% RSLogix 500 project LEGACY PROGRAM NO LABELS ORIGINAL_BAK006.RSS, saved by version 11.00.00.00 %
PROJECT "ML1200"    % processor: MicroLogix 1200; MAIN_PROG %

PROGRAM FILES
  LAD 2 "MAIN_PROG"  15 rungs
  LAD 3   18 rungs
  LAD 4   33 rungs
  LAD 5   12 rungs
  LAD 6   14 rungs
  LAD 7   2 rungs
  LAD 8   47 rungs
  LAD 9   2 rungs
  LAD 10   5 rungs
  LAD 11   14 rungs

DATA FILES
  O0 OUTPUT  8 elements
  I1 INPUT  19 elements
  S2 STATUS  66 elements
  B3 BINARY  20 elements
  T4 TIMER  13 elements
  C5 COUNTER  1 elements
  R6 CONTROL  1 elements
  N7 INTEGER  77 elements
  F8 FLOAT  1 elements
  PD9   3 elements

LADDER 2 "MAIN_PROG"
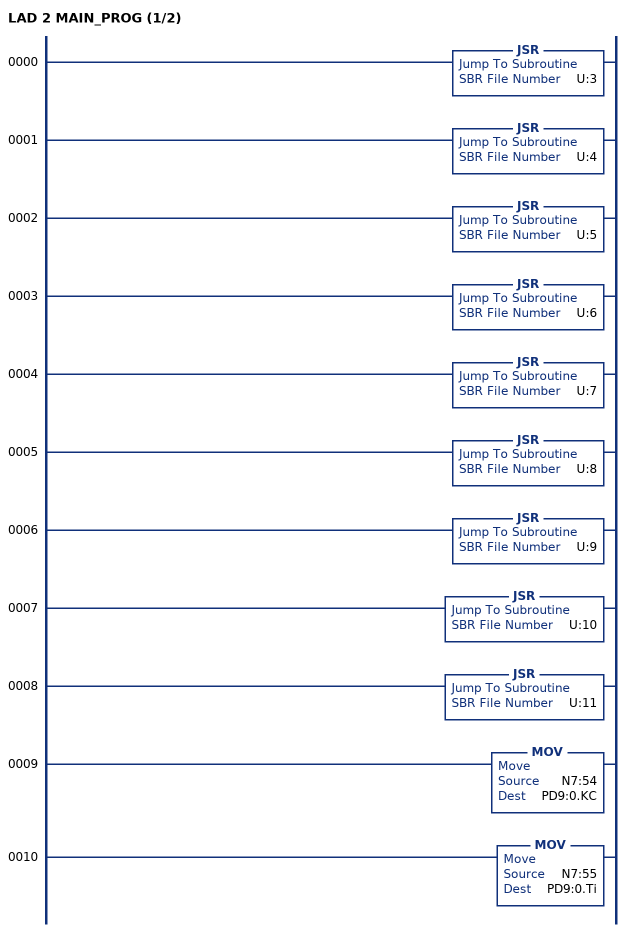
% Rung: 0 %
SOR JSR U:3 EOR
% Rung: 1 %
SOR JSR U:4 EOR
% Rung: 2 %
SOR JSR U:5 EOR
% Rung: 3 %
SOR JSR U:6 EOR
% Rung: 4 %
SOR JSR U:7 EOR
% Rung: 5 %
SOR JSR U:8 EOR
% Rung: 6 %
SOR JSR U:9 EOR
% Rung: 7 %
SOR JSR U:10 EOR
% Rung: 8 %
SOR JSR U:11 EOR
% Rung: 9 %
SOR MOV N7:54 PD9:0.KC EOR
% Rung: 10 %
SOR MOV N7:55 PD9:0.Ti EOR

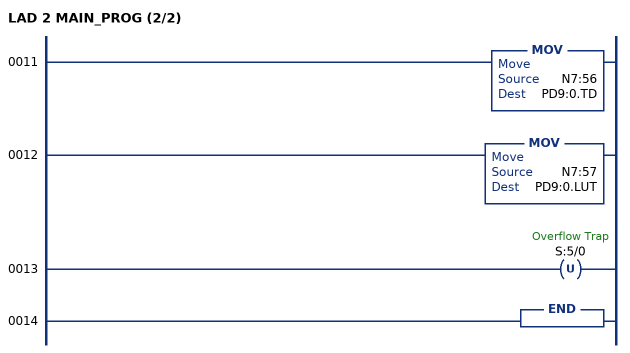
% Rung: 11 %
SOR MOV N7:56 PD9:0.TD EOR
% Rung: 12 %
SOR MOV N7:57 PD9:0.LUT EOR
% Rung: 13 %
SOR OTU S:5/0 EOR
%   S:5/0  "Overflow Trap" %
% Rung: 14 %
SOR END EOR

LADDER 3
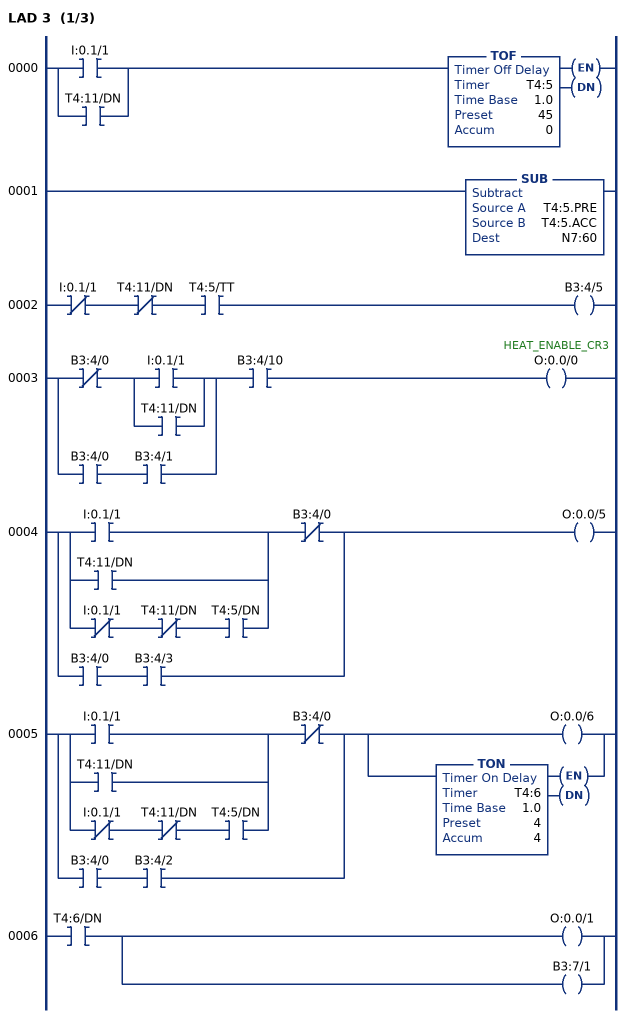
% Rung: 0 %
SOR BST XIC I:0.1/1 NXB XIC T4:11/DN BND TOF T4:5 1.0 45 0 EOR
% Rung: 1 %
SOR SUB T4:5.PRE T4:5.ACC N7:60 EOR
% Rung: 2 %
SOR XIO I:0.1/1 XIO T4:11/DN XIC T4:5/TT OTE B3:4/5 EOR
% Rung: 3 %
SOR BST XIO B3:4/0 BST XIC I:0.1/1 NXB XIC T4:11/DN BND NXB XIC B3:4/0 XIC B3:4/1 BND XIC B3:4/10 OTE O:0.0/0 EOR
%   O:0.0/0  HEAT_ENABLE_CR3 %
% Rung: 4 %
SOR BST BST BST XIC I:0.1/1 NXB XIC T4:11/DN BND NXB XIO I:0.1/1 XIO T4:11/DN XIC T4:5/DN BND XIO B3:4/0 NXB XIC B3:4/0 XIC B3:4/3 BND OTE O:0.0/5 EOR
% Rung: 5 %
SOR BST BST BST XIC I:0.1/1 NXB XIC T4:11/DN BND NXB XIO I:0.1/1 XIO T4:11/DN XIC T4:5/DN BND XIO B3:4/0 NXB XIC B3:4/0 XIC B3:4/2 BND BST OTE O:0.0/6 NXB TON T4:6 1.0 4 4 BND EOR
% Rung: 6 %
SOR XIC T4:6/DN BST OTE O:0.0/1 NXB OTE B3:7/1 BND EOR

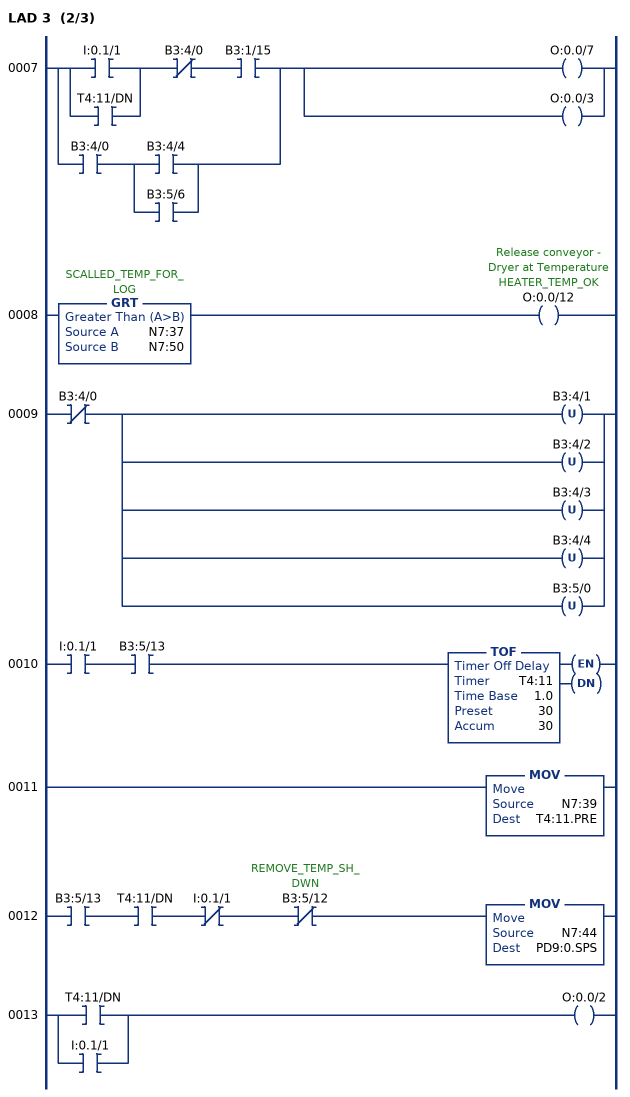
% Rung: 7 %
SOR BST BST XIC I:0.1/1 NXB XIC T4:11/DN BND XIO B3:4/0 XIC B3:1/15 NXB XIC B3:4/0 BST XIC B3:4/4 NXB XIC B3:5/6 BND BND BST OTE O:0.0/7 NXB OTE O:0.0/3 BND EOR
% Rung: 8 %
SOR GRT N7:37 N7:50 OTE O:0.0/12 EOR
%   N7:37  SCALLED_TEMP_FOR_LOG %
%   N7:50  CONVEYOR_REASE_TEMP %
%   O:0.0/12  HEATER_TEMP_OK  "Release conveyor - Dryer at Temperature" %
% Rung: 9 %
SOR XIO B3:4/0 BST OTU B3:4/1 NXB BST OTU B3:4/2 NXB BST OTU B3:4/3 NXB BST OTU B3:4/4 NXB OTU B3:5/0 BND BND BND BND EOR
% Rung: 10 %
SOR XIC I:0.1/1 XIC B3:5/13 TOF T4:11 1.0 30 30 EOR
% Rung: 11 %
SOR MOV N7:39 T4:11.PRE EOR
% Rung: 12 %
SOR XIC B3:5/13 XIC T4:11/DN XIO I:0.1/1 XIO B3:5/12 MOV N7:44 PD9:0.SPS EOR
%   B3:5/12  REMOVE_TEMP_SH_DWN %
% Rung: 13 %
SOR BST XIC T4:11/DN NXB XIC I:0.1/1 BND OTE O:0.0/2 EOR

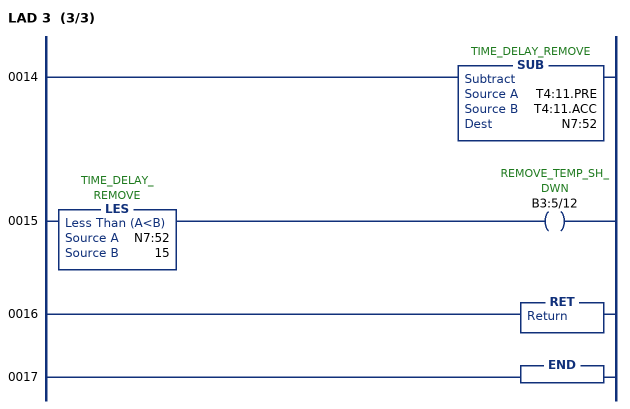
% Rung: 14 %
SOR SUB T4:11.PRE T4:11.ACC N7:52 EOR
%   N7:52  TIME_DELAY_REMOVE %
% Rung: 15 %
SOR LES N7:52 15 OTE B3:5/12 EOR
%   N7:52  TIME_DELAY_REMOVE %
%   B3:5/12  REMOVE_TEMP_SH_DWN %
% Rung: 16 %
SOR RET EOR
% Rung: 17 %
SOR END EOR

LADDER 4
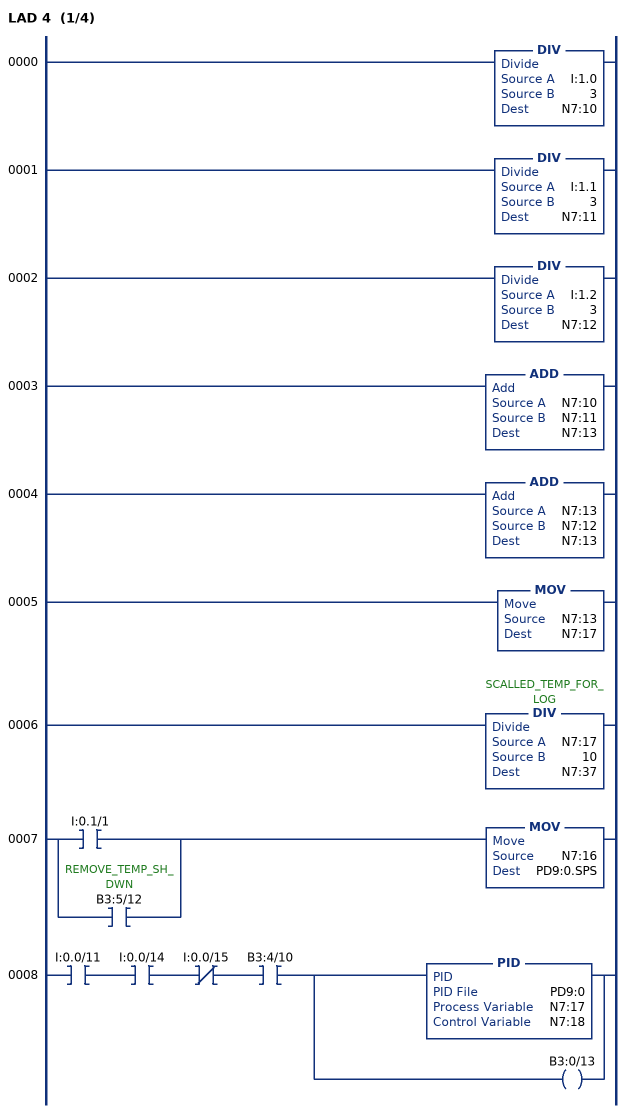
% Rung: 0 %
SOR DIV I:1.0 3 N7:10 EOR
% Rung: 1 %
SOR DIV I:1.1 3 N7:11 EOR
% Rung: 2 %
SOR DIV I:1.2 3 N7:12 EOR
% Rung: 3 %
SOR ADD N7:10 N7:11 N7:13 EOR
% Rung: 4 %
SOR ADD N7:13 N7:12 N7:13 EOR
% Rung: 5 %
SOR MOV N7:13 N7:17 EOR
% Rung: 6 %
SOR DIV N7:17 10 N7:37 EOR
%   N7:37  SCALLED_TEMP_FOR_LOG %
% Rung: 7 %
SOR BST XIC I:0.1/1 NXB XIC B3:5/12 BND MOV N7:16 PD9:0.SPS EOR
%   B3:5/12  REMOVE_TEMP_SH_DWN %
% Rung: 8 %
SOR XIC I:0.0/11 XIC I:0.0/14 XIO I:0.0/15 XIC B3:4/10 BST PID PD9:0 N7:17 N7:18 NXB OTE B3:0/13 BND EOR

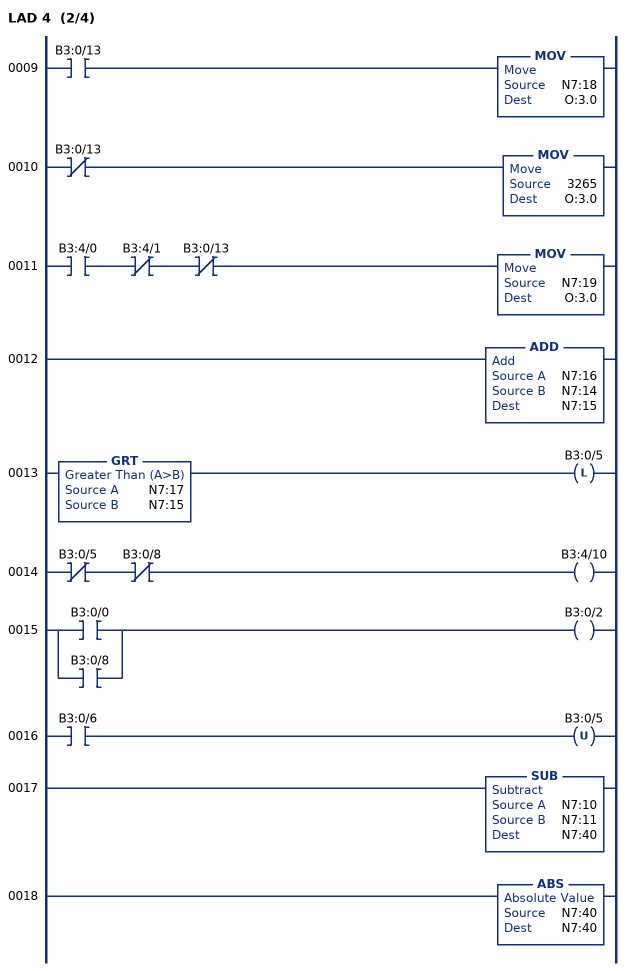
% Rung: 9 %
SOR XIC B3:0/13 MOV N7:18 O:3.0 EOR
% Rung: 10 %
SOR XIO B3:0/13 MOV 3265 O:3.0 EOR
% Rung: 11 %
SOR XIC B3:4/0 XIO B3:4/1 XIO B3:0/13 MOV N7:19 O:3.0 EOR
% Rung: 12 %
SOR ADD N7:16 N7:14 N7:15 EOR
% Rung: 13 %
SOR GRT N7:17 N7:15 OTL B3:0/5 EOR
% Rung: 14 %
SOR XIO B3:0/5 XIO B3:0/8 OTE B3:4/10 EOR
% Rung: 15 %
SOR BST XIC B3:0/0 NXB XIC B3:0/8 BND OTE B3:0/2 EOR
% Rung: 16 %
SOR XIC B3:0/6 OTU B3:0/5 EOR
% Rung: 17 %
SOR SUB N7:10 N7:11 N7:40 EOR
% Rung: 18 %
SOR ABS N7:40 N7:40 EOR

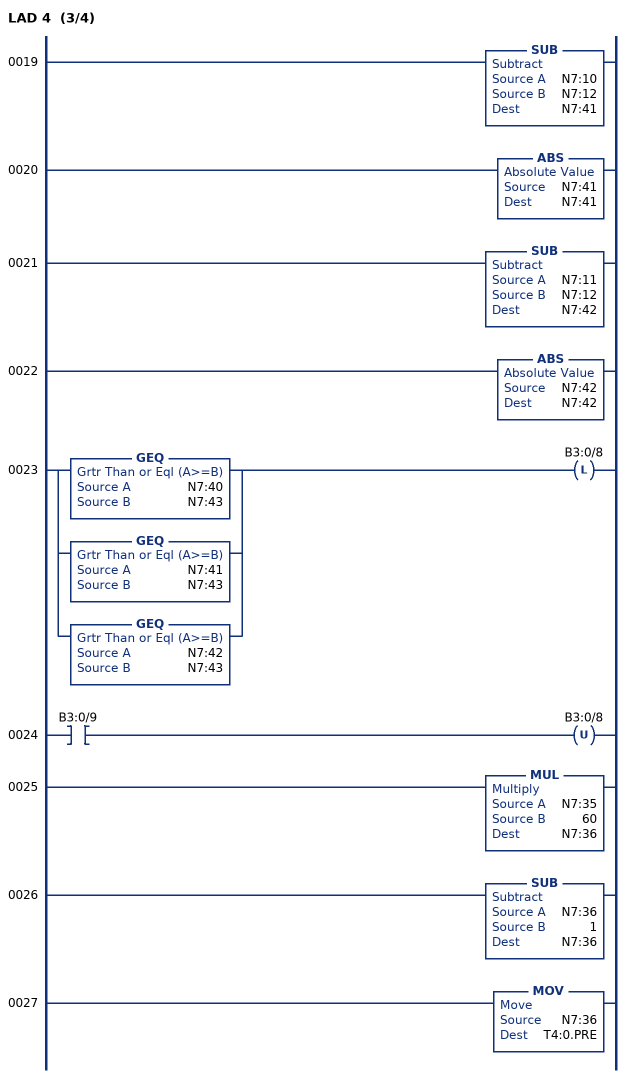
% Rung: 19 %
SOR SUB N7:10 N7:12 N7:41 EOR
% Rung: 20 %
SOR ABS N7:41 N7:41 EOR
% Rung: 21 %
SOR SUB N7:11 N7:12 N7:42 EOR
% Rung: 22 %
SOR ABS N7:42 N7:42 EOR
% Rung: 23 %
SOR BST GEQ N7:40 N7:43 NXB BST GEQ N7:41 N7:43 NXB GEQ N7:42 N7:43 BND BND OTL B3:0/8 EOR
% Rung: 24 %
SOR XIC B3:0/9 OTU B3:0/8 EOR
% Rung: 25 %
SOR MUL N7:35 60 N7:36 EOR
% Rung: 26 %
SOR SUB N7:36 1 N7:36 EOR
% Rung: 27 %
SOR MOV N7:36 T4:0.PRE EOR

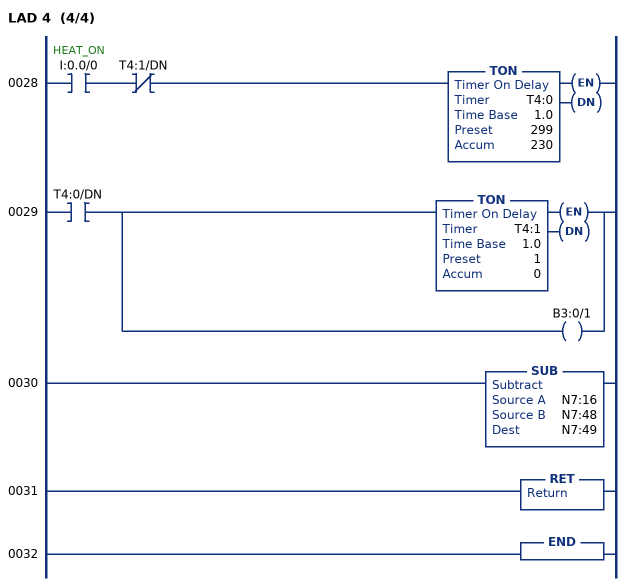
% Rung: 28 %
SOR XIC I:0.0/0 XIO T4:1/DN TON T4:0 1.0 299 230 EOR
%   I:0.0/0  HEAT_ON %
% Rung: 29 %
SOR XIC T4:0/DN BST TON T4:1 1.0 1 0 NXB OTE B3:0/1 BND EOR
% Rung: 30 %
SOR SUB N7:16 N7:48 N7:49 EOR
% Rung: 31 %
SOR RET EOR
% Rung: 32 %
SOR END EOR

LADDER 5
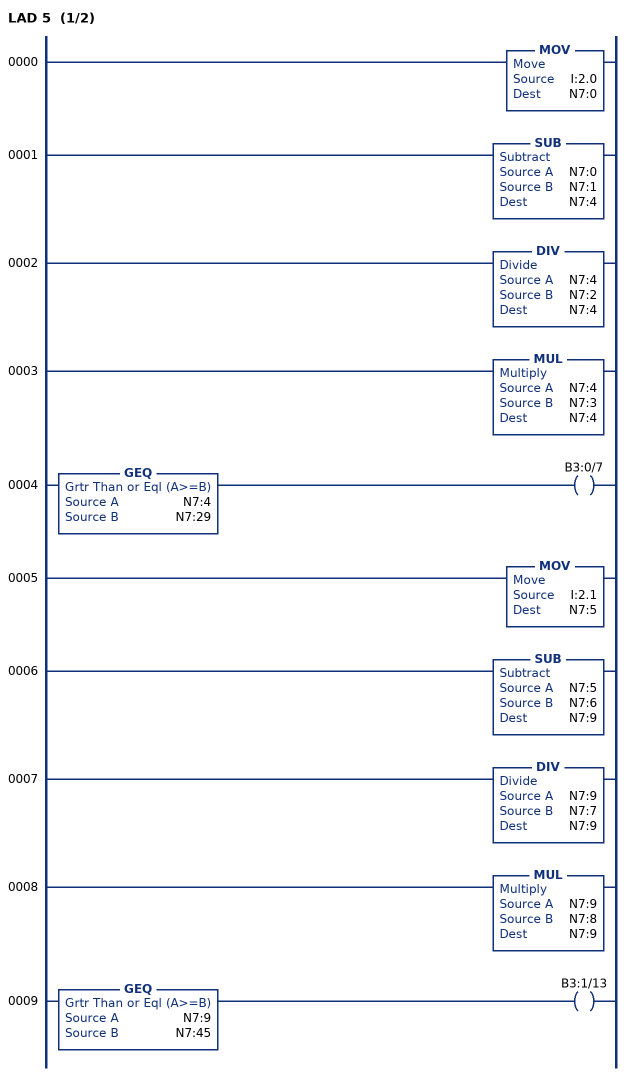
% Rung: 0 %
SOR MOV I:2.0 N7:0 EOR
% Rung: 1 %
SOR SUB N7:0 N7:1 N7:4 EOR
% Rung: 2 %
SOR DIV N7:4 N7:2 N7:4 EOR
% Rung: 3 %
SOR MUL N7:4 N7:3 N7:4 EOR
% Rung: 4 %
SOR GEQ N7:4 N7:29 OTE B3:0/7 EOR
% Rung: 5 %
SOR MOV I:2.1 N7:5 EOR
% Rung: 6 %
SOR SUB N7:5 N7:6 N7:9 EOR
% Rung: 7 %
SOR DIV N7:9 N7:7 N7:9 EOR
% Rung: 8 %
SOR MUL N7:9 N7:8 N7:9 EOR
% Rung: 9 %
SOR GEQ N7:9 N7:45 OTE B3:1/13 EOR

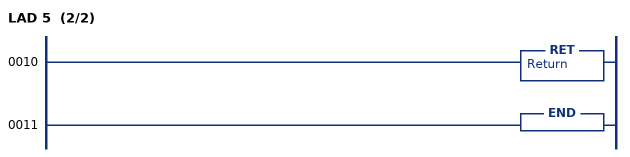
% Rung: 10 %
SOR RET EOR
% Rung: 11 %
SOR END EOR

LADDER 6
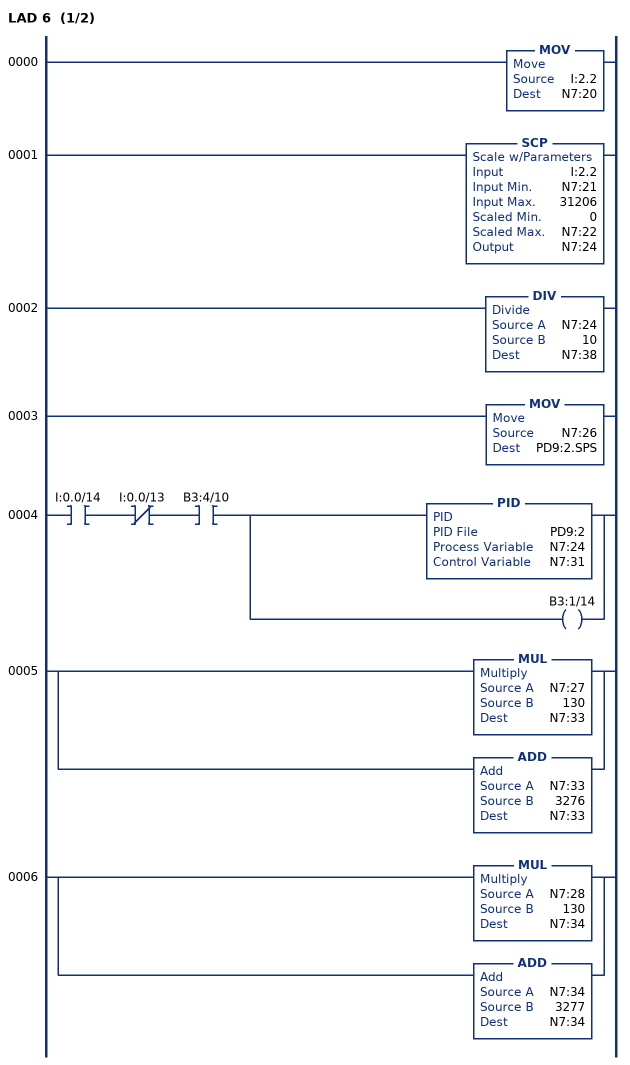
% Rung: 0 %
SOR MOV I:2.2 N7:20 EOR
% Rung: 1 %
SOR SCP I:2.2 N7:21 31206 0 N7:22 N7:24 EOR
% Rung: 2 %
SOR DIV N7:24 10 N7:38 EOR
% Rung: 3 %
SOR MOV N7:26 PD9:2.SPS EOR
% Rung: 4 %
SOR XIC I:0.0/14 XIO I:0.0/13 XIC B3:4/10 BST PID PD9:2 N7:24 N7:31 NXB OTE B3:1/14 BND EOR
% Rung: 5 %
SOR BST MUL N7:27 130 N7:33 NXB ADD N7:33 3276 N7:33 BND EOR
% Rung: 6 %
SOR BST MUL N7:28 130 N7:34 NXB ADD N7:34 3277 N7:34 BND EOR

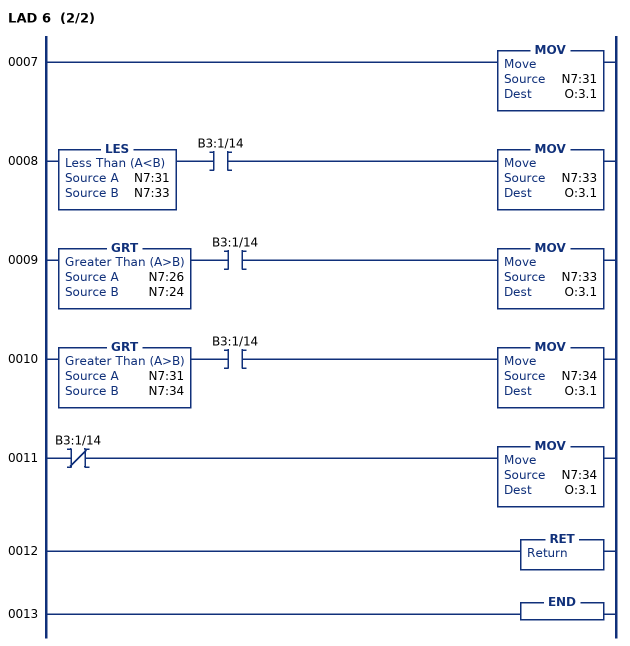
% Rung: 7 %
SOR MOV N7:31 O:3.1 EOR
% Rung: 8 %
SOR LES N7:31 N7:33 XIC B3:1/14 MOV N7:33 O:3.1 EOR
% Rung: 9 %
SOR GRT N7:26 N7:24 XIC B3:1/14 MOV N7:33 O:3.1 EOR
% Rung: 10 %
SOR GRT N7:31 N7:34 XIC B3:1/14 MOV N7:34 O:3.1 EOR
% Rung: 11 %
SOR XIO B3:1/14 MOV N7:34 O:3.1 EOR
% Rung: 12 %
SOR RET EOR
% Rung: 13 %
SOR END EOR

LADDER 7
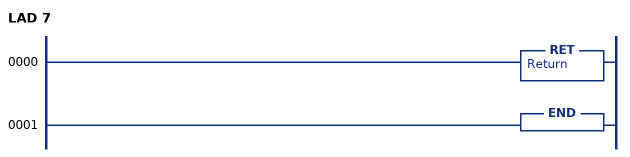
% Rung: 0 %
SOR RET EOR
% Rung: 1 %
SOR END EOR

LADDER 8
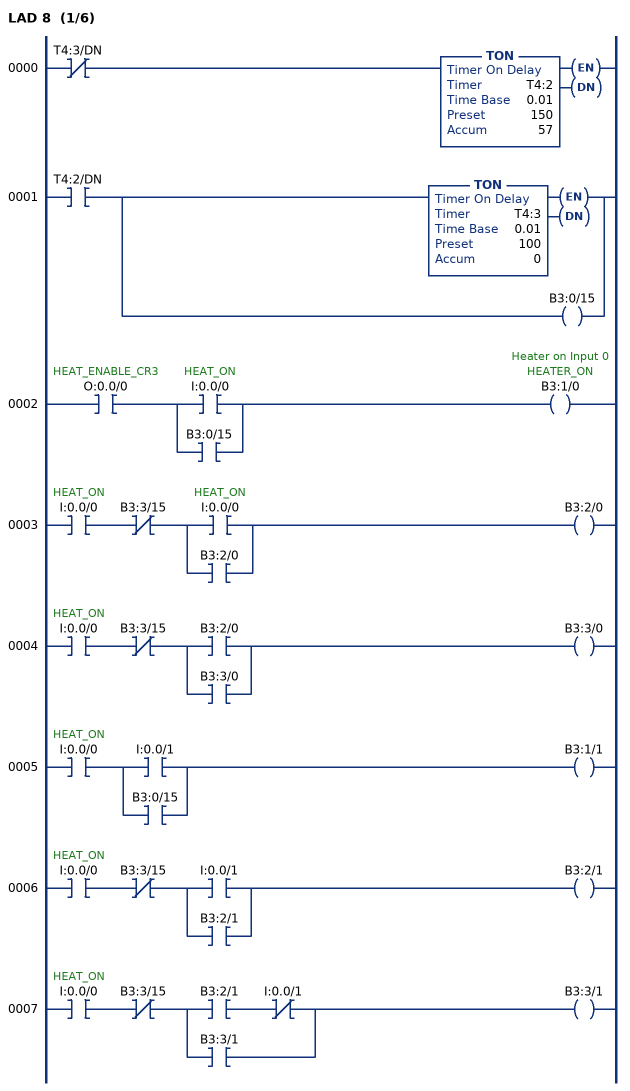
% Rung: 0 %
SOR XIO T4:3/DN TON T4:2 0.01 150 57 EOR
% Rung: 1 %
SOR XIC T4:2/DN BST TON T4:3 0.01 100 0 NXB OTE B3:0/15 BND EOR
% Rung: 2 %
SOR XIC O:0.0/0 BST XIC I:0.0/0 NXB XIC B3:0/15 BND OTE B3:1/0 EOR
%   O:0.0/0  HEAT_ENABLE_CR3 %
%   I:0.0/0  HEAT_ON %
%   B3:1/0  HEATER_ON  "Heater on Input 0" %
% Rung: 3 %
SOR XIC I:0.0/0 XIO B3:3/15 BST XIC I:0.0/0 NXB XIC B3:2/0 BND OTE B3:2/0 EOR
%   I:0.0/0  HEAT_ON %
% Rung: 4 %
SOR XIC I:0.0/0 XIO B3:3/15 BST XIC B3:2/0 NXB XIC B3:3/0 BND OTE B3:3/0 EOR
%   I:0.0/0  HEAT_ON %
% Rung: 5 %
SOR XIC I:0.0/0 BST XIC I:0.0/1 NXB XIC B3:0/15 BND OTE B3:1/1 EOR
%   I:0.0/0  HEAT_ON %
% Rung: 6 %
SOR XIC I:0.0/0 XIO B3:3/15 BST XIC I:0.0/1 NXB XIC B3:2/1 BND OTE B3:2/1 EOR
%   I:0.0/0  HEAT_ON %
% Rung: 7 %
SOR XIC I:0.0/0 XIO B3:3/15 BST XIC B3:2/1 XIO I:0.0/1 NXB XIC B3:3/1 BND OTE B3:3/1 EOR
%   I:0.0/0  HEAT_ON %

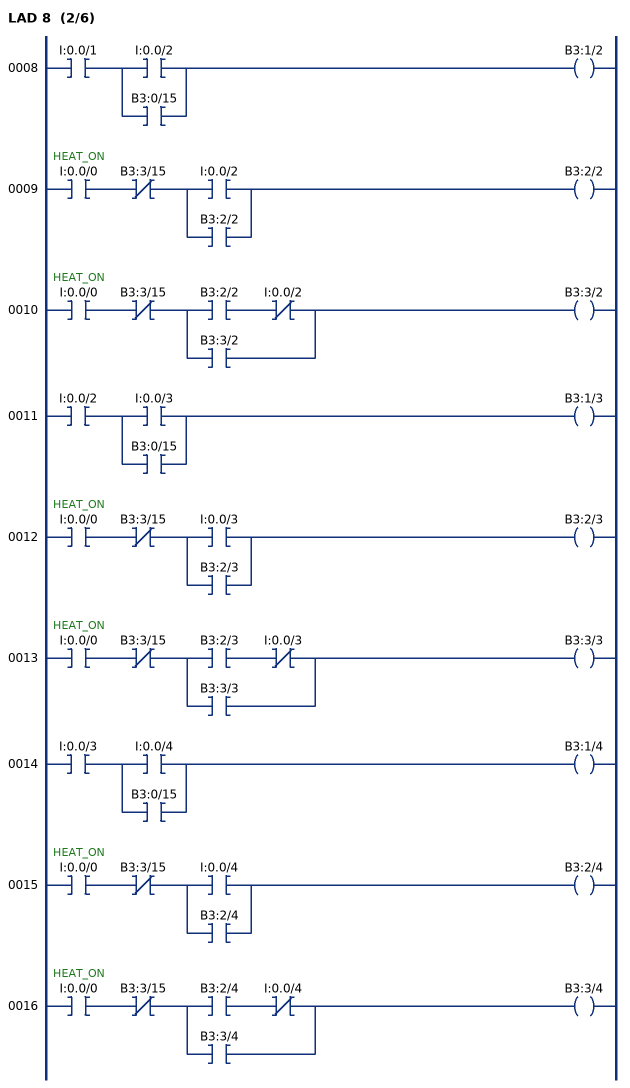
% Rung: 8 %
SOR XIC I:0.0/1 BST XIC I:0.0/2 NXB XIC B3:0/15 BND OTE B3:1/2 EOR
% Rung: 9 %
SOR XIC I:0.0/0 XIO B3:3/15 BST XIC I:0.0/2 NXB XIC B3:2/2 BND OTE B3:2/2 EOR
%   I:0.0/0  HEAT_ON %
% Rung: 10 %
SOR XIC I:0.0/0 XIO B3:3/15 BST XIC B3:2/2 XIO I:0.0/2 NXB XIC B3:3/2 BND OTE B3:3/2 EOR
%   I:0.0/0  HEAT_ON %
% Rung: 11 %
SOR XIC I:0.0/2 BST XIC I:0.0/3 NXB XIC B3:0/15 BND OTE B3:1/3 EOR
% Rung: 12 %
SOR XIC I:0.0/0 XIO B3:3/15 BST XIC I:0.0/3 NXB XIC B3:2/3 BND OTE B3:2/3 EOR
%   I:0.0/0  HEAT_ON %
% Rung: 13 %
SOR XIC I:0.0/0 XIO B3:3/15 BST XIC B3:2/3 XIO I:0.0/3 NXB XIC B3:3/3 BND OTE B3:3/3 EOR
%   I:0.0/0  HEAT_ON %
% Rung: 14 %
SOR XIC I:0.0/3 BST XIC I:0.0/4 NXB XIC B3:0/15 BND OTE B3:1/4 EOR
% Rung: 15 %
SOR XIC I:0.0/0 XIO B3:3/15 BST XIC I:0.0/4 NXB XIC B3:2/4 BND OTE B3:2/4 EOR
%   I:0.0/0  HEAT_ON %
% Rung: 16 %
SOR XIC I:0.0/0 XIO B3:3/15 BST XIC B3:2/4 XIO I:0.0/4 NXB XIC B3:3/4 BND OTE B3:3/4 EOR
%   I:0.0/0  HEAT_ON %

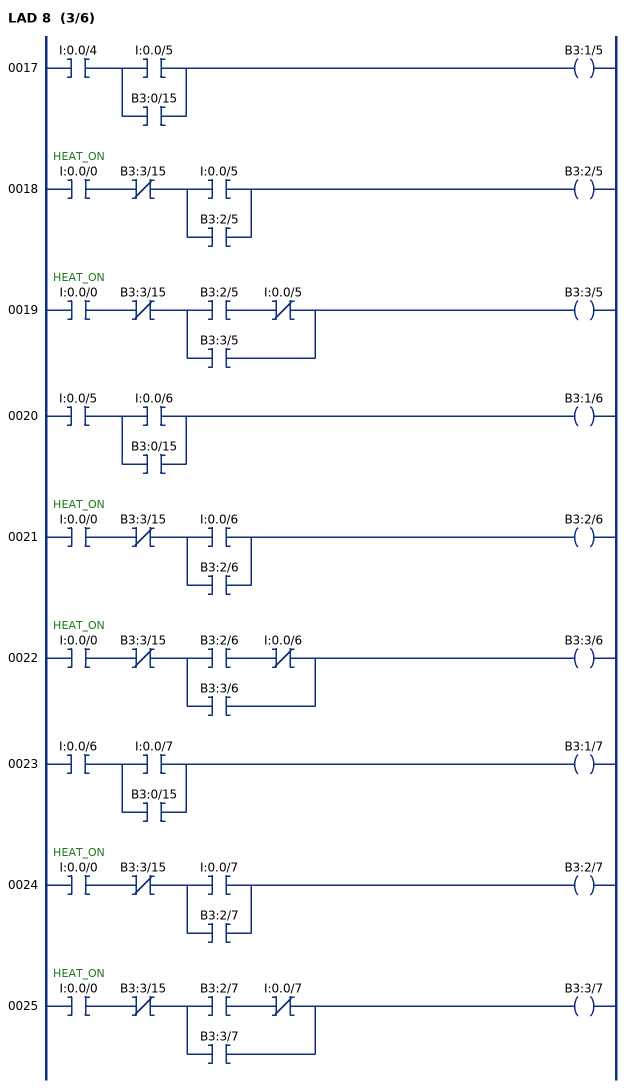
% Rung: 17 %
SOR XIC I:0.0/4 BST XIC I:0.0/5 NXB XIC B3:0/15 BND OTE B3:1/5 EOR
% Rung: 18 %
SOR XIC I:0.0/0 XIO B3:3/15 BST XIC I:0.0/5 NXB XIC B3:2/5 BND OTE B3:2/5 EOR
%   I:0.0/0  HEAT_ON %
% Rung: 19 %
SOR XIC I:0.0/0 XIO B3:3/15 BST XIC B3:2/5 XIO I:0.0/5 NXB XIC B3:3/5 BND OTE B3:3/5 EOR
%   I:0.0/0  HEAT_ON %
% Rung: 20 %
SOR XIC I:0.0/5 BST XIC I:0.0/6 NXB XIC B3:0/15 BND OTE B3:1/6 EOR
% Rung: 21 %
SOR XIC I:0.0/0 XIO B3:3/15 BST XIC I:0.0/6 NXB XIC B3:2/6 BND OTE B3:2/6 EOR
%   I:0.0/0  HEAT_ON %
% Rung: 22 %
SOR XIC I:0.0/0 XIO B3:3/15 BST XIC B3:2/6 XIO I:0.0/6 NXB XIC B3:3/6 BND OTE B3:3/6 EOR
%   I:0.0/0  HEAT_ON %
% Rung: 23 %
SOR XIC I:0.0/6 BST XIC I:0.0/7 NXB XIC B3:0/15 BND OTE B3:1/7 EOR
% Rung: 24 %
SOR XIC I:0.0/0 XIO B3:3/15 BST XIC I:0.0/7 NXB XIC B3:2/7 BND OTE B3:2/7 EOR
%   I:0.0/0  HEAT_ON %
% Rung: 25 %
SOR XIC I:0.0/0 XIO B3:3/15 BST XIC B3:2/7 XIO I:0.0/7 NXB XIC B3:3/7 BND OTE B3:3/7 EOR
%   I:0.0/0  HEAT_ON %

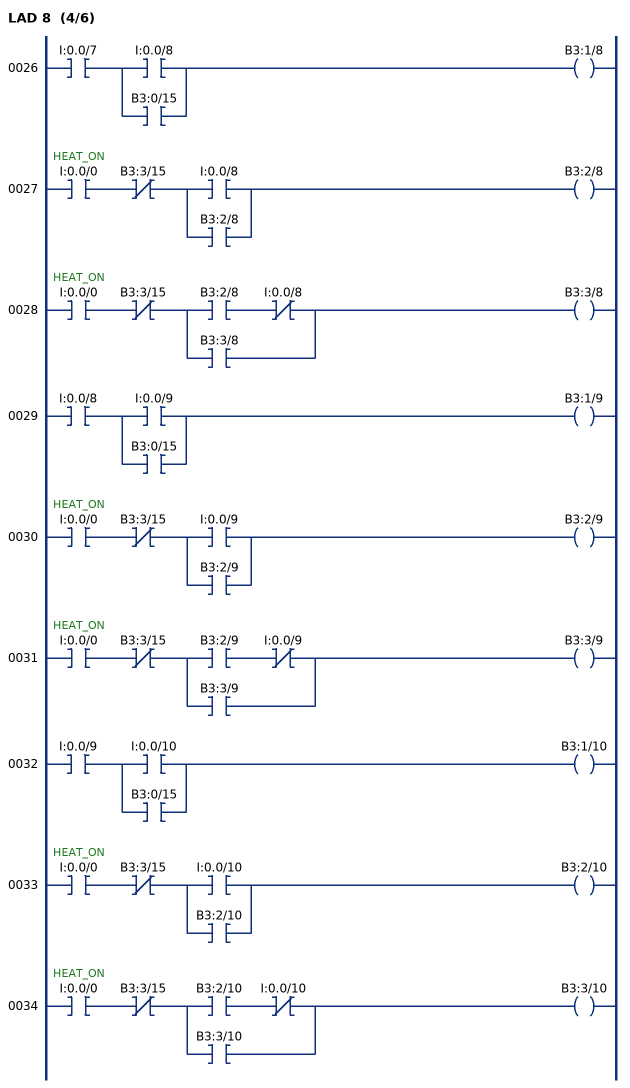
% Rung: 26 %
SOR XIC I:0.0/7 BST XIC I:0.0/8 NXB XIC B3:0/15 BND OTE B3:1/8 EOR
% Rung: 27 %
SOR XIC I:0.0/0 XIO B3:3/15 BST XIC I:0.0/8 NXB XIC B3:2/8 BND OTE B3:2/8 EOR
%   I:0.0/0  HEAT_ON %
% Rung: 28 %
SOR XIC I:0.0/0 XIO B3:3/15 BST XIC B3:2/8 XIO I:0.0/8 NXB XIC B3:3/8 BND OTE B3:3/8 EOR
%   I:0.0/0  HEAT_ON %
% Rung: 29 %
SOR XIC I:0.0/8 BST XIC I:0.0/9 NXB XIC B3:0/15 BND OTE B3:1/9 EOR
% Rung: 30 %
SOR XIC I:0.0/0 XIO B3:3/15 BST XIC I:0.0/9 NXB XIC B3:2/9 BND OTE B3:2/9 EOR
%   I:0.0/0  HEAT_ON %
% Rung: 31 %
SOR XIC I:0.0/0 XIO B3:3/15 BST XIC B3:2/9 XIO I:0.0/9 NXB XIC B3:3/9 BND OTE B3:3/9 EOR
%   I:0.0/0  HEAT_ON %
% Rung: 32 %
SOR XIC I:0.0/9 BST XIC I:0.0/10 NXB XIC B3:0/15 BND OTE B3:1/10 EOR
% Rung: 33 %
SOR XIC I:0.0/0 XIO B3:3/15 BST XIC I:0.0/10 NXB XIC B3:2/10 BND OTE B3:2/10 EOR
%   I:0.0/0  HEAT_ON %
% Rung: 34 %
SOR XIC I:0.0/0 XIO B3:3/15 BST XIC B3:2/10 XIO I:0.0/10 NXB XIC B3:3/10 BND OTE B3:3/10 EOR
%   I:0.0/0  HEAT_ON %

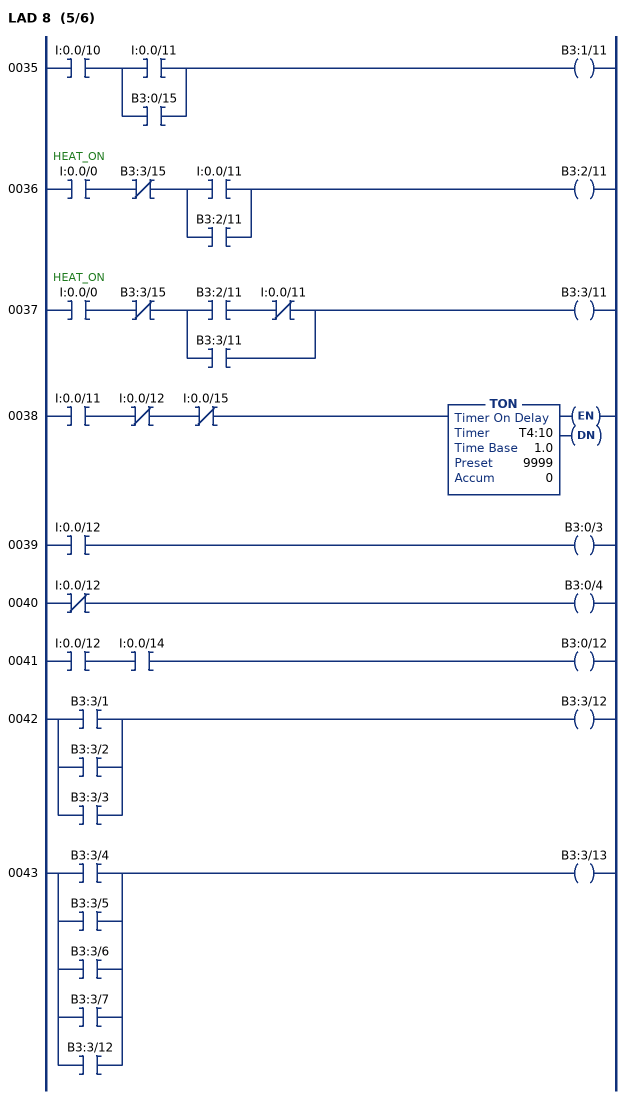
% Rung: 35 %
SOR XIC I:0.0/10 BST XIC I:0.0/11 NXB XIC B3:0/15 BND OTE B3:1/11 EOR
% Rung: 36 %
SOR XIC I:0.0/0 XIO B3:3/15 BST XIC I:0.0/11 NXB XIC B3:2/11 BND OTE B3:2/11 EOR
%   I:0.0/0  HEAT_ON %
% Rung: 37 %
SOR XIC I:0.0/0 XIO B3:3/15 BST XIC B3:2/11 XIO I:0.0/11 NXB XIC B3:3/11 BND OTE B3:3/11 EOR
%   I:0.0/0  HEAT_ON %
% Rung: 38 %
SOR XIC I:0.0/11 XIO I:0.0/12 XIO I:0.0/15 TON T4:10 1.0 9999 0 EOR
% Rung: 39 %
SOR XIC I:0.0/12 OTE B3:0/3 EOR
% Rung: 40 %
SOR XIO I:0.0/12 OTE B3:0/4 EOR
% Rung: 41 %
SOR XIC I:0.0/12 XIC I:0.0/14 OTE B3:0/12 EOR
% Rung: 42 %
SOR BST XIC B3:3/1 NXB BST XIC B3:3/2 NXB XIC B3:3/3 BND BND OTE B3:3/12 EOR
% Rung: 43 %
SOR BST XIC B3:3/4 NXB BST XIC B3:3/5 NXB BST XIC B3:3/6 NXB BST XIC B3:3/7 NXB XIC B3:3/12 BND BND BND BND OTE B3:3/13 EOR

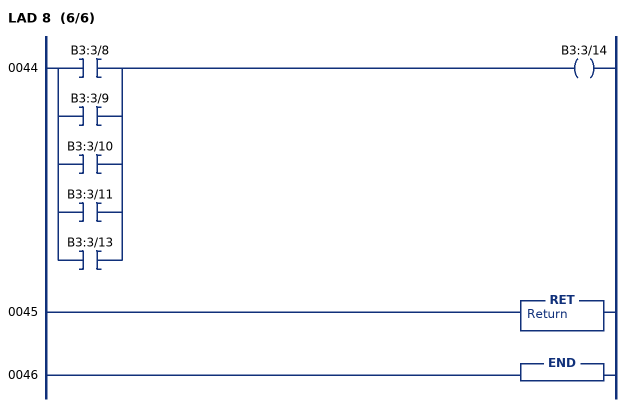
% Rung: 44 %
SOR BST XIC B3:3/8 NXB BST XIC B3:3/9 NXB BST XIC B3:3/10 NXB BST XIC B3:3/11 NXB XIC B3:3/13 BND BND BND BND OTE B3:3/14 EOR
% Rung: 45 %
SOR RET EOR
% Rung: 46 %
SOR END EOR

LADDER 9
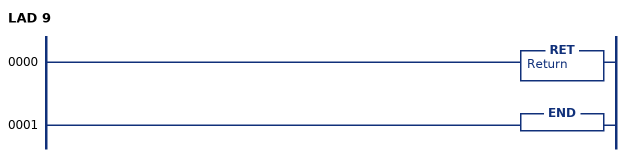
% Rung: 0 %
SOR RET EOR
% Rung: 1 %
SOR END EOR

LADDER 10
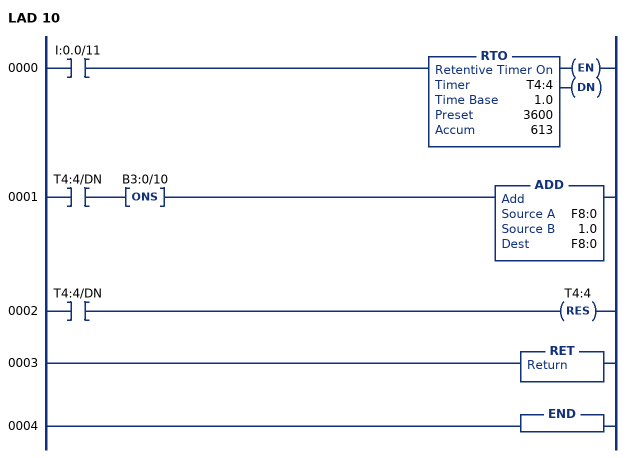
% Rung: 0 %
SOR XIC I:0.0/11 RTO T4:4 1.0 3600 613 EOR
% Rung: 1 %
SOR XIC T4:4/DN ONS B3:0/10 ADD F8:0 1.0 F8:0 EOR
% Rung: 2 %
SOR XIC T4:4/DN RES T4:4 EOR
% Rung: 3 %
SOR RET EOR
% Rung: 4 %
SOR END EOR

LADDER 11
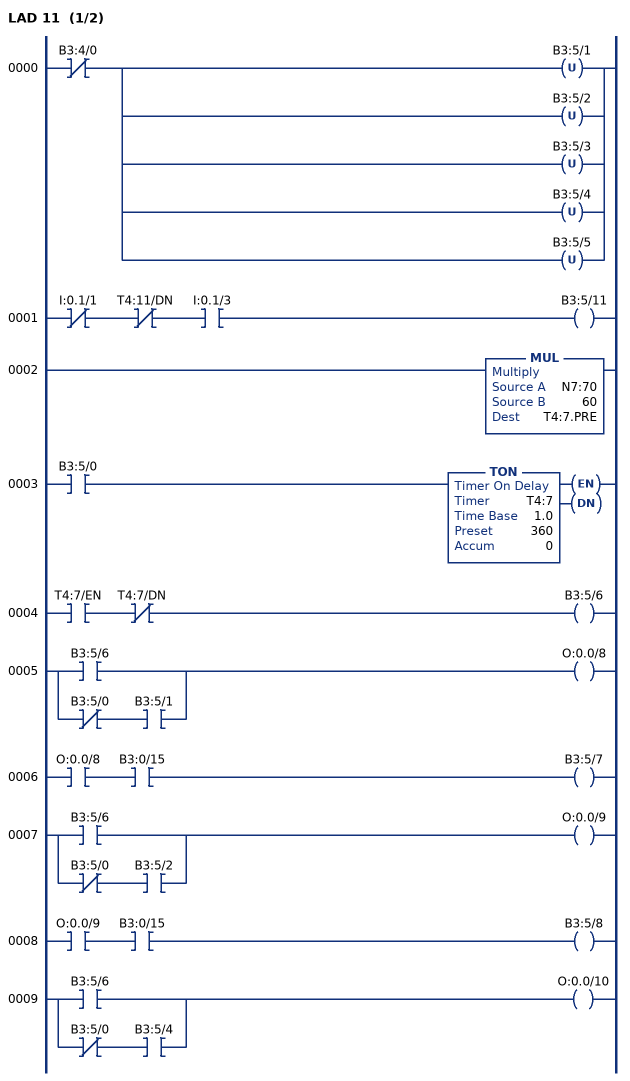
% Rung: 0 %
SOR XIO B3:4/0 BST OTU B3:5/1 NXB BST OTU B3:5/2 NXB BST OTU B3:5/3 NXB BST OTU B3:5/4 NXB OTU B3:5/5 BND BND BND BND EOR
% Rung: 1 %
SOR XIO I:0.1/1 XIO T4:11/DN XIC I:0.1/3 OTE B3:5/11 EOR
% Rung: 2 %
SOR MUL N7:70 60 T4:7.PRE EOR
% Rung: 3 %
SOR XIC B3:5/0 TON T4:7 1.0 360 0 EOR
% Rung: 4 %
SOR XIC T4:7/EN XIO T4:7/DN OTE B3:5/6 EOR
% Rung: 5 %
SOR BST XIC B3:5/6 NXB XIO B3:5/0 XIC B3:5/1 BND OTE O:0.0/8 EOR
% Rung: 6 %
SOR XIC O:0.0/8 XIC B3:0/15 OTE B3:5/7 EOR
% Rung: 7 %
SOR BST XIC B3:5/6 NXB XIO B3:5/0 XIC B3:5/2 BND OTE O:0.0/9 EOR
% Rung: 8 %
SOR XIC O:0.0/9 XIC B3:0/15 OTE B3:5/8 EOR
% Rung: 9 %
SOR BST XIC B3:5/6 NXB XIO B3:5/0 XIC B3:5/4 BND OTE O:0.0/10 EOR

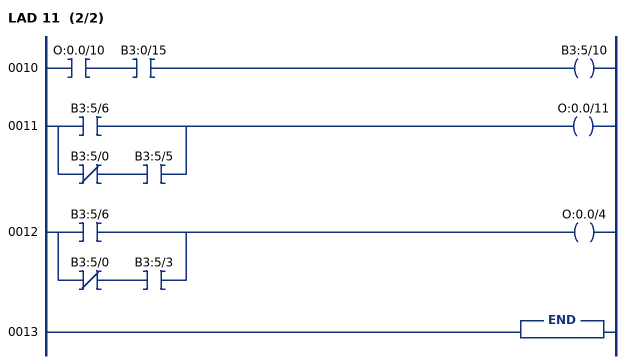
% Rung: 10 %
SOR XIC O:0.0/10 XIC B3:0/15 OTE B3:5/10 EOR
% Rung: 11 %
SOR BST XIC B3:5/6 NXB XIO B3:5/0 XIC B3:5/5 BND OTE O:0.0/11 EOR
% Rung: 12 %
SOR BST XIC B3:5/6 NXB XIO B3:5/0 XIC B3:5/3 BND OTE O:0.0/4 EOR
% Rung: 13 %
SOR END EOR

DATA TABLE (non-zero values as saved)
DATA B3
% B3:0 % 0X3008 0XCFFF 0X0FFF 0X0001 0X0580 0X0000 0X0000 0X0102 0X0000 0X0000
% B3:10 % 0X0001 0X0000 0X0000 0X0000 0X0000 0X0000 0X0000 0X0000 0X0000 0X0000
DATA T4
% .PRE .ACC %
% T4:0 % 299 230
% T4:1 % 1 0
% T4:2 % 150 57
% T4:3 % 100 0
% T4:4 % 3600 613
% T4:5 % 45 0
% T4:6 % 4 4
% T4:7 % 360 0
% T4:8 % 600 0
% T4:9 % 1800 0
% T4:10 % 9999 0
% T4:11 % 30 30
% T4:12 % 30 20
DATA N7
% N7:0 % 6956 6226 105 1 7 6280 6265 18 1 1
% N7:10 % 450 448 451 1349 300 1650 1350 1349 11572 3400
% N7:20 % 8968 6250 240 10 26 25 5 60 100 12
% N7:30 % 10 0 195 11076 16277 5 299 135 3 30
% N7:40 % 2 1 3 200 1200 5 0 0 0 1350
% N7:50 % 85 10 0 0 60 1 20 20 0 0
% N7:60 % 45 0 0 0 0 0 0 0 0 0
% N7:70 % 6 0 0 0 0 0 0
DATA F8
% F8:0 % 14
